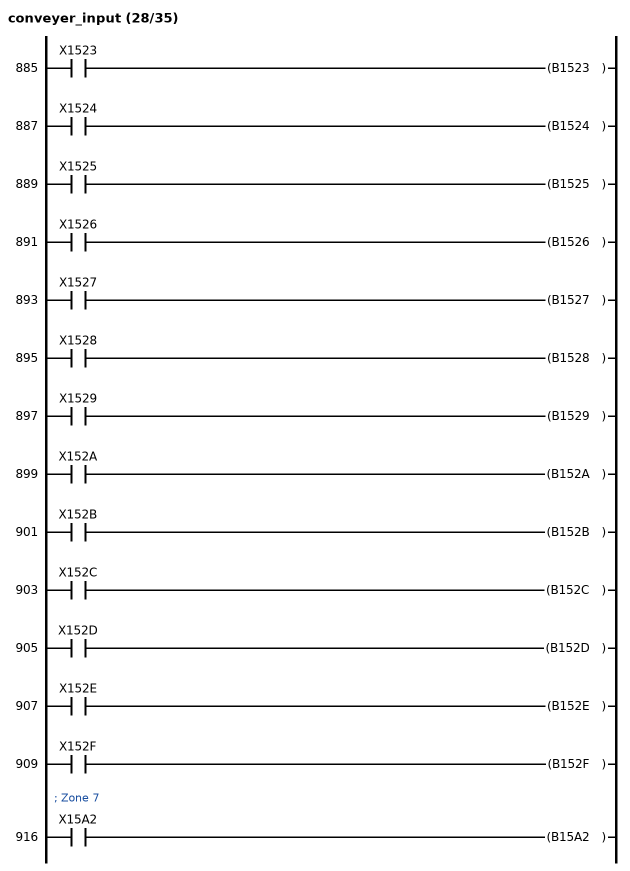
[picture p120: ladder of conveyer_input, rungs at steps 885 to 916]
885   LD      X1523
      OUT     B1523
887   LD      X1524
      OUT     B1524
889   LD      X1525
      OUT     B1525
891   LD      X1526
      OUT     B1526
893   LD      X1527
      OUT     B1527
895   LD      X1528
      OUT     B1528
897   LD      X1529
      OUT     B1529
899   LD      X152A
      OUT     B152A
901   LD      X152B
      OUT     B152B
903   LD      X152C
      OUT     B152C
905   LD      X152D
      OUT     B152D
907   LD      X152E
      OUT     B152E
909   LD      X152F
      OUT     B152F
; Zone 7
916   LD      X15A2
      OUT     B15A2
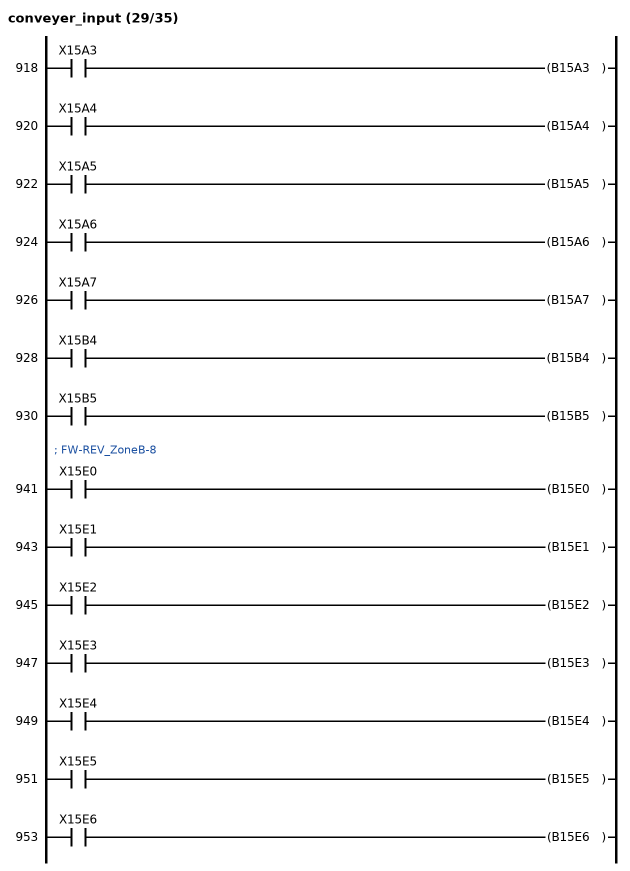
918   LD      X15A3
      OUT     B15A3
920   LD      X15A4
      OUT     B15A4
922   LD      X15A5
      OUT     B15A5
924   LD      X15A6
      OUT     B15A6
926   LD      X15A7
      OUT     B15A7
928   LD      X15B4
      OUT     B15B4
930   LD      X15B5
      OUT     B15B5
; FW-REV_ZoneB-8
941   LD      X15E0
      OUT     B15E0
943   LD      X15E1
      OUT     B15E1
945   LD      X15E2
      OUT     B15E2
947   LD      X15E3
      OUT     B15E3
949   LD      X15E4
      OUT     B15E4
951   LD      X15E5
      OUT     B15E5
953   LD      X15E6
      OUT     B15E6
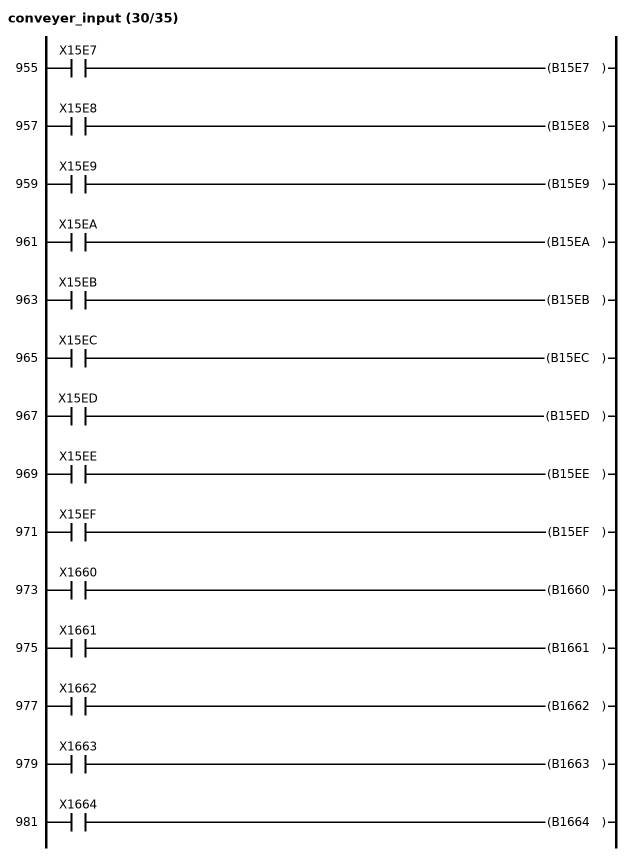
955   LD      X15E7
      OUT     B15E7
957   LD      X15E8
      OUT     B15E8
959   LD      X15E9
      OUT     B15E9
961   LD      X15EA
      OUT     B15EA
963   LD      X15EB
      OUT     B15EB
965   LD      X15EC
      OUT     B15EC
967   LD      X15ED
      OUT     B15ED
969   LD      X15EE
      OUT     B15EE
971   LD      X15EF
      OUT     B15EF
973   LD      X1660
      OUT     B1660
975   LD      X1661
      OUT     B1661
977   LD      X1662
      OUT     B1662
979   LD      X1663
      OUT     B1663
981   LD      X1664
      OUT     B1664
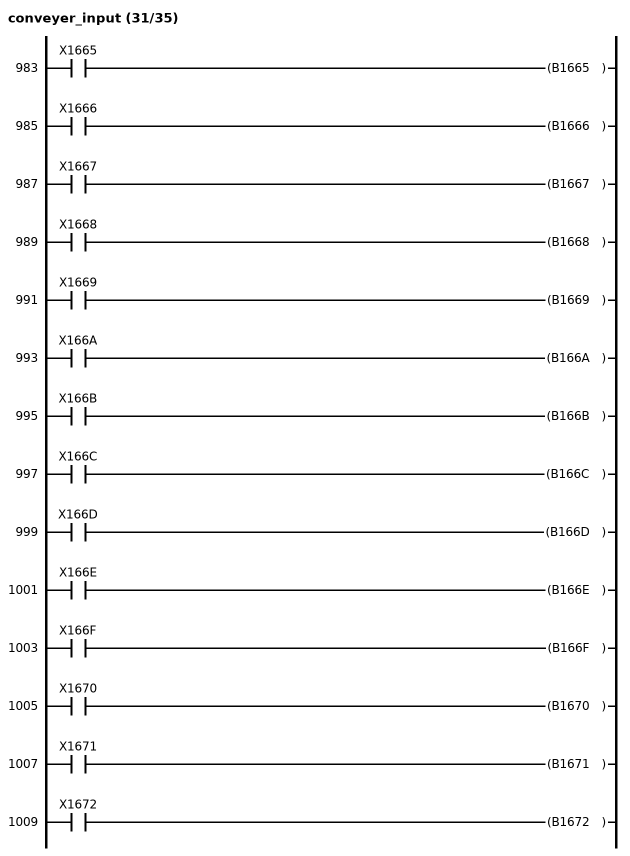
983   LD      X1665
      OUT     B1665
985   LD      X1666
      OUT     B1666
987   LD      X1667
      OUT     B1667
989   LD      X1668
      OUT     B1668
991   LD      X1669
      OUT     B1669
993   LD      X166A
      OUT     B166A
995   LD      X166B
      OUT     B166B
997   LD      X166C
      OUT     B166C
999   LD      X166D
      OUT     B166D
1001  LD      X166E
      OUT     B166E
1003  LD      X166F
      OUT     B166F
1005  LD      X1670
      OUT     B1670
1007  LD      X1671
      OUT     B1671
1009  LD      X1672
      OUT     B1672
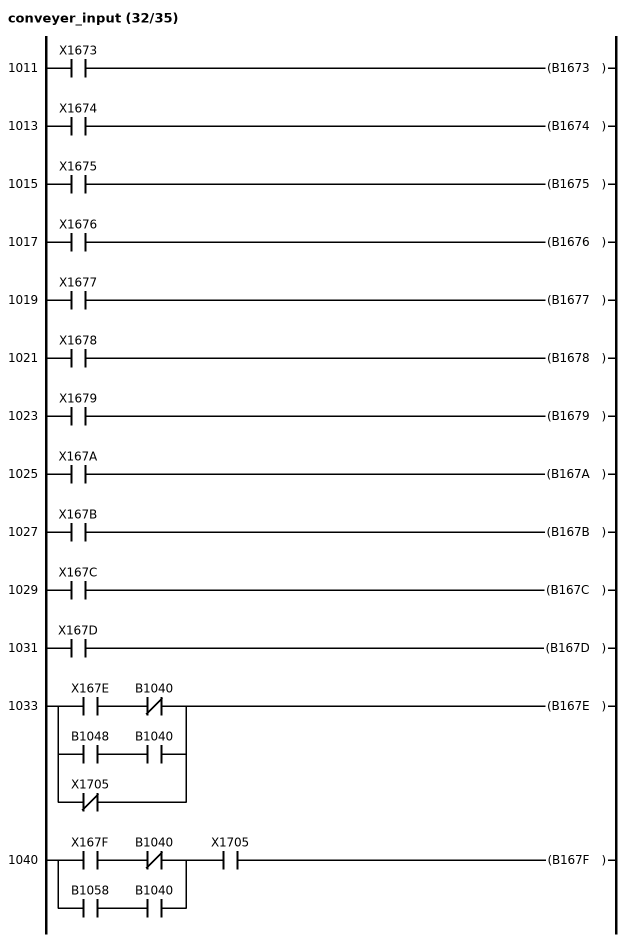
1011  LD      X1673
      OUT     B1673
1013  LD      X1674
      OUT     B1674
1015  LD      X1675
      OUT     B1675
1017  LD      X1676
      OUT     B1676
1019  LD      X1677
      OUT     B1677
1021  LD      X1678
      OUT     B1678
1023  LD      X1679
      OUT     B1679
1025  LD      X167A
      OUT     B167A
1027  LD      X167B
      OUT     B167B
1029  LD      X167C
      OUT     B167C
1031  LD      X167D
      OUT     B167D
1033  LD      X167E
      ANI     B1040
      LD      B1048
      AND     B1040
      ORB
      ORI     X1705
      OUT     B167E
1040  LD      X167F
      ANI     B1040
      LD      B1058
      AND     B1040
      ORB
      AND     X1705
      OUT     B167F
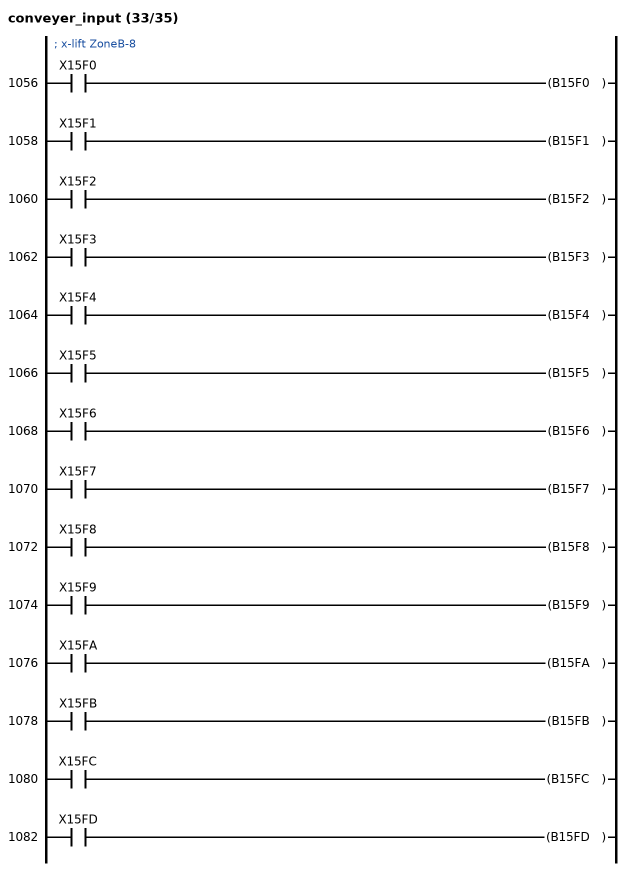
; x-lift ZoneB-8
1056  LD      X15F0
      OUT     B15F0
1058  LD      X15F1
      OUT     B15F1
1060  LD      X15F2
      OUT     B15F2
1062  LD      X15F3
      OUT     B15F3
1064  LD      X15F4
      OUT     B15F4
1066  LD      X15F5
      OUT     B15F5
1068  LD      X15F6
      OUT     B15F6
1070  LD      X15F7
      OUT     B15F7
1072  LD      X15F8
      OUT     B15F8
1074  LD      X15F9
      OUT     B15F9
1076  LD      X15FA
      OUT     B15FA
1078  LD      X15FB
      OUT     B15FB
1080  LD      X15FC
      OUT     B15FC
1082  LD      X15FD
      OUT     B15FD
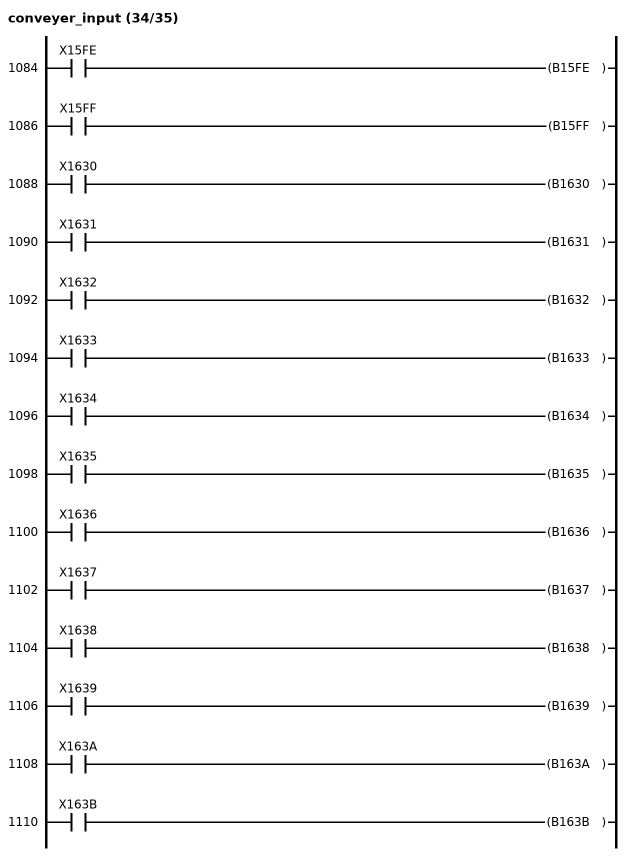
1084  LD      X15FE
      OUT     B15FE
1086  LD      X15FF
      OUT     B15FF
1088  LD      X1630
      OUT     B1630
1090  LD      X1631
      OUT     B1631
1092  LD      X1632
      OUT     B1632
1094  LD      X1633
      OUT     B1633
1096  LD      X1634
      OUT     B1634
1098  LD      X1635
      OUT     B1635
1100  LD      X1636
      OUT     B1636
1102  LD      X1637
      OUT     B1637
1104  LD      X1638
      OUT     B1638
1106  LD      X1639
      OUT     B1639
1108  LD      X163A
      OUT     B163A
1110  LD      X163B
      OUT     B163B
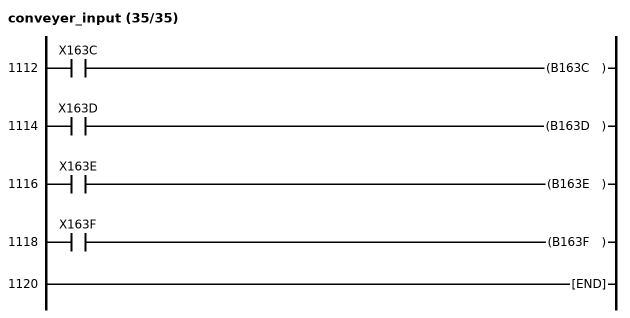
1112  LD      X163C
      OUT     B163C
1114  LD      X163D
      OUT     B163D
1116  LD      X163E
      OUT     B163E
1118  LD      X163F
      OUT     B163F
1120  END
END_PROGRAM

PROGRAM conveyor_output
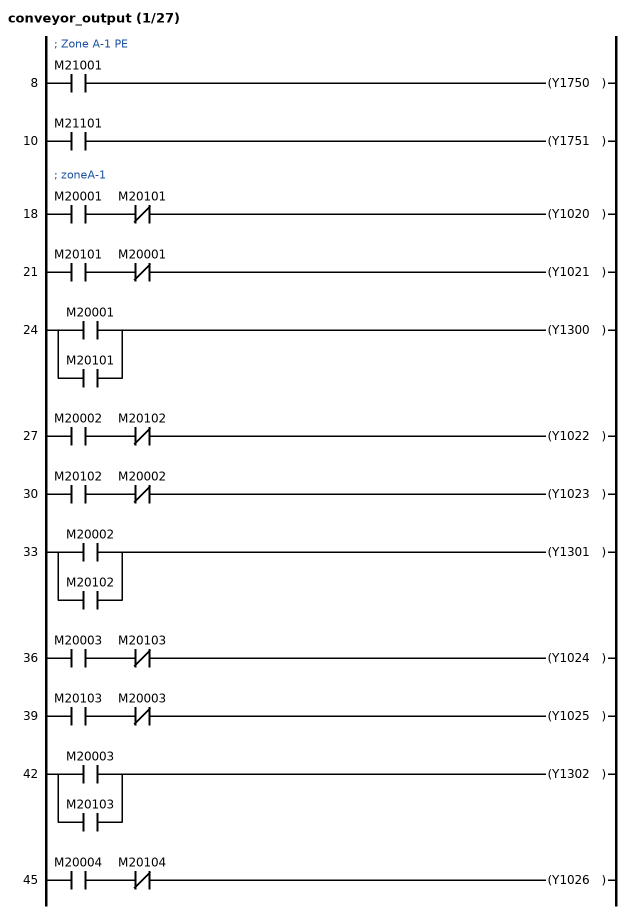
; Zone A-1 PE
8     LD      M21001
      OUT     Y1750
10    LD      M21101
      OUT     Y1751
; zoneA-1
18    LD      M20001
      ANI     M20101
      OUT     Y1020
21    LD      M20101
      ANI     M20001
      OUT     Y1021
24    LD      M20001
      OR      M20101
      OUT     Y1300
27    LD      M20002
      ANI     M20102
      OUT     Y1022
30    LD      M20102
      ANI     M20002
      OUT     Y1023
33    LD      M20002
      OR      M20102
      OUT     Y1301
36    LD      M20003
      ANI     M20103
      OUT     Y1024
39    LD      M20103
      ANI     M20003
      OUT     Y1025
42    LD      M20003
      OR      M20103
      OUT     Y1302
45    LD      M20004
      ANI     M20104
      OUT     Y1026
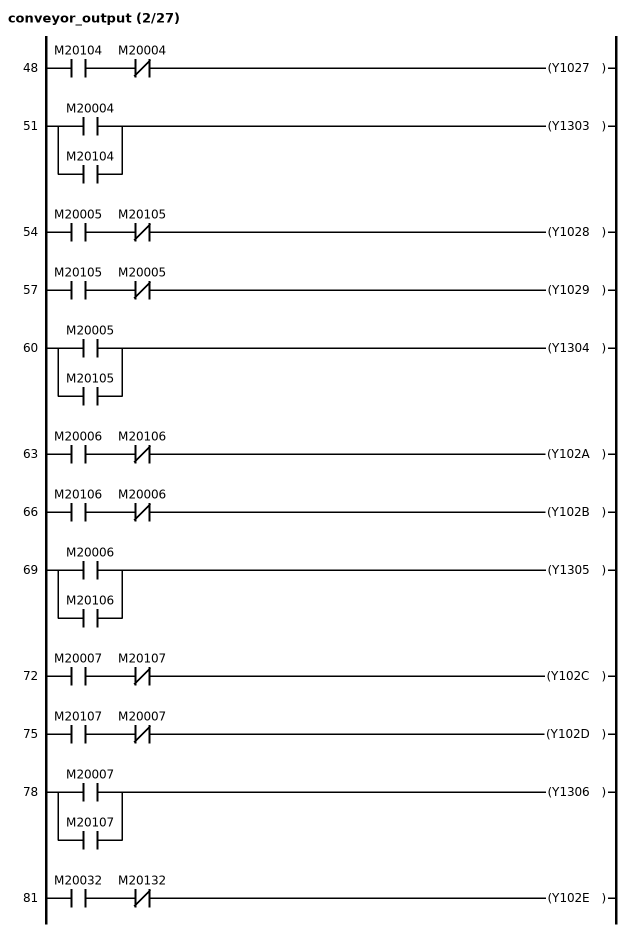
48    LD      M20104
      ANI     M20004
      OUT     Y1027
51    LD      M20004
      OR      M20104
      OUT     Y1303
54    LD      M20005
      ANI     M20105
      OUT     Y1028
57    LD      M20105
      ANI     M20005
      OUT     Y1029
60    LD      M20005
      OR      M20105
      OUT     Y1304
63    LD      M20006
      ANI     M20106
      OUT     Y102A
66    LD      M20106
      ANI     M20006
      OUT     Y102B
69    LD      M20006
      OR      M20106
      OUT     Y1305
72    LD      M20007
      ANI     M20107
      OUT     Y102C
75    LD      M20107
      ANI     M20007
      OUT     Y102D
78    LD      M20007
      OR      M20107
      OUT     Y1306
81    LD      M20032
      ANI     M20132
      OUT     Y102E
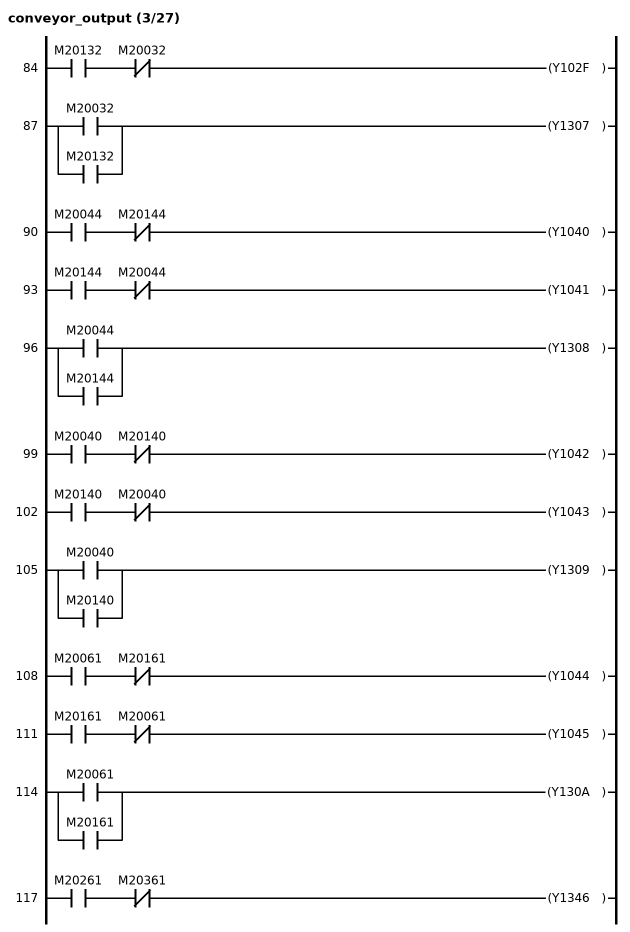
84    LD      M20132
      ANI     M20032
      OUT     Y102F
87    LD      M20032
      OR      M20132
      OUT     Y1307
90    LD      M20044
      ANI     M20144
      OUT     Y1040
93    LD      M20144
      ANI     M20044
      OUT     Y1041
96    LD      M20044
      OR      M20144
      OUT     Y1308
99    LD      M20040
      ANI     M20140
      OUT     Y1042
102   LD      M20140
      ANI     M20040
      OUT     Y1043
105   LD      M20040
      OR      M20140
      OUT     Y1309
108   LD      M20061
      ANI     M20161
      OUT     Y1044
111   LD      M20161
      ANI     M20061
      OUT     Y1045
114   LD      M20061
      OR      M20161
      OUT     Y130A
117   LD      M20261
      ANI     M20361
      OUT     Y1346
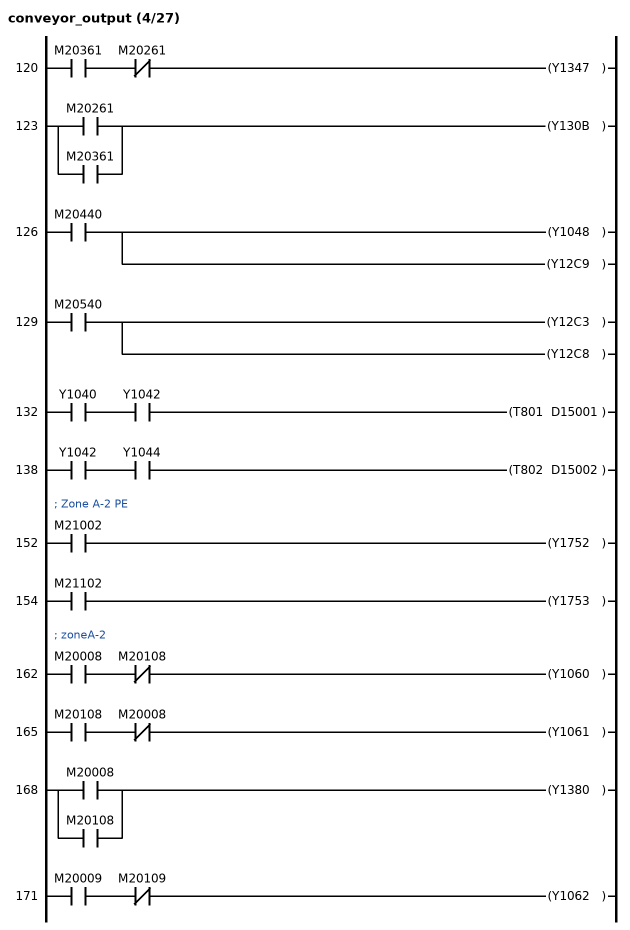
120   LD      M20361
      ANI     M20261
      OUT     Y1347
123   LD      M20261
      OR      M20361
      OUT     Y130B
126   LD      M20440
      OUT     Y1048
      OUT     Y12C9
129   LD      M20540
      OUT     Y12C3
      OUT     Y12C8
132   LD      Y1040
      AND     Y1042
      OUT     T801 D15001
138   LD      Y1042
      AND     Y1044
      OUT     T802 D15002
; Zone A-2 PE
152   LD      M21002
      OUT     Y1752
154   LD      M21102
      OUT     Y1753
; zoneA-2
162   LD      M20008
      ANI     M20108
      OUT     Y1060
165   LD      M20108
      ANI     M20008
      OUT     Y1061
168   LD      M20008
      OR      M20108
      OUT     Y1380
171   LD      M20009
      ANI     M20109
      OUT     Y1062
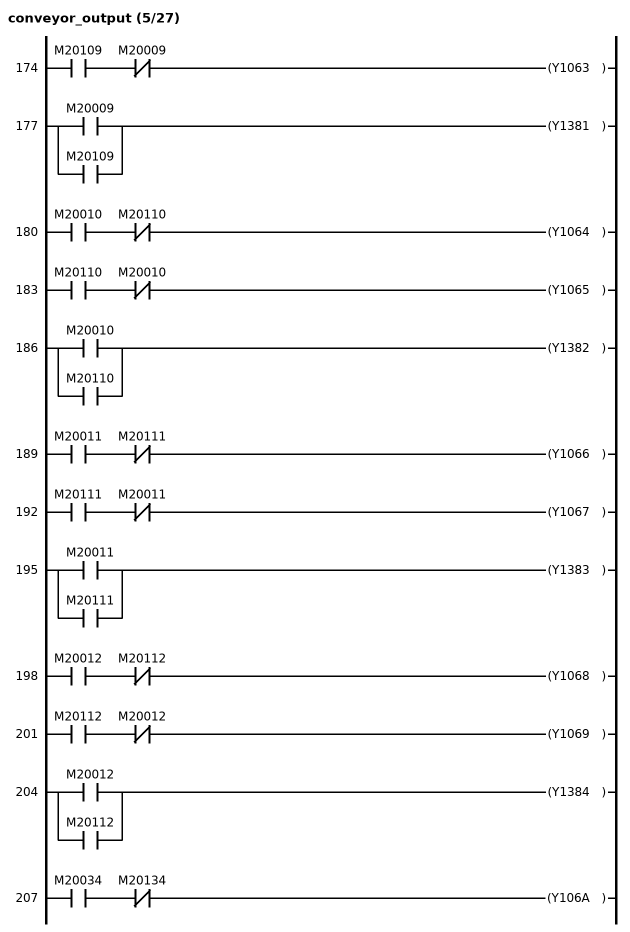
174   LD      M20109
      ANI     M20009
      OUT     Y1063
177   LD      M20009
      OR      M20109
      OUT     Y1381
180   LD      M20010
      ANI     M20110
      OUT     Y1064
183   LD      M20110
      ANI     M20010
      OUT     Y1065
186   LD      M20010
      OR      M20110
      OUT     Y1382
189   LD      M20011
      ANI     M20111
      OUT     Y1066
192   LD      M20111
      ANI     M20011
      OUT     Y1067
195   LD      M20011
      OR      M20111
      OUT     Y1383
198   LD      M20012
      ANI     M20112
      OUT     Y1068
201   LD      M20112
      ANI     M20012
      OUT     Y1069
204   LD      M20012
      OR      M20112
      OUT     Y1384
207   LD      M20034
      ANI     M20134
      OUT     Y106A
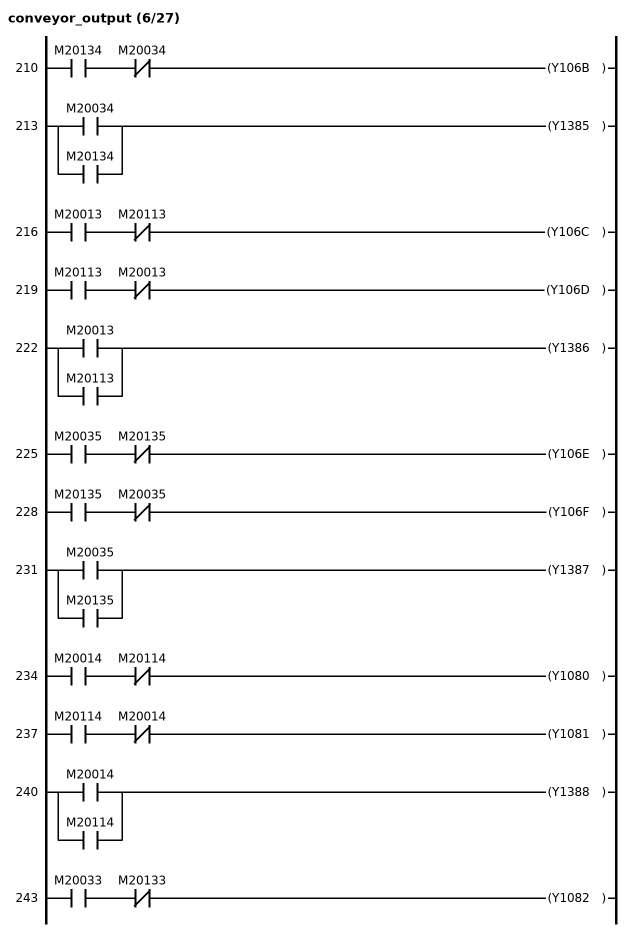
210   LD      M20134
      ANI     M20034
      OUT     Y106B
213   LD      M20034
      OR      M20134
      OUT     Y1385
216   LD      M20013
      ANI     M20113
      OUT     Y106C
219   LD      M20113
      ANI     M20013
      OUT     Y106D
222   LD      M20013
      OR      M20113
      OUT     Y1386
225   LD      M20035
      ANI     M20135
      OUT     Y106E
228   LD      M20135
      ANI     M20035
      OUT     Y106F
231   LD      M20035
      OR      M20135
      OUT     Y1387
234   LD      M20014
      ANI     M20114
      OUT     Y1080
237   LD      M20114
      ANI     M20014
      OUT     Y1081
240   LD      M20014
      OR      M20114
      OUT     Y1388
243   LD      M20033
      ANI     M20133
      OUT     Y1082
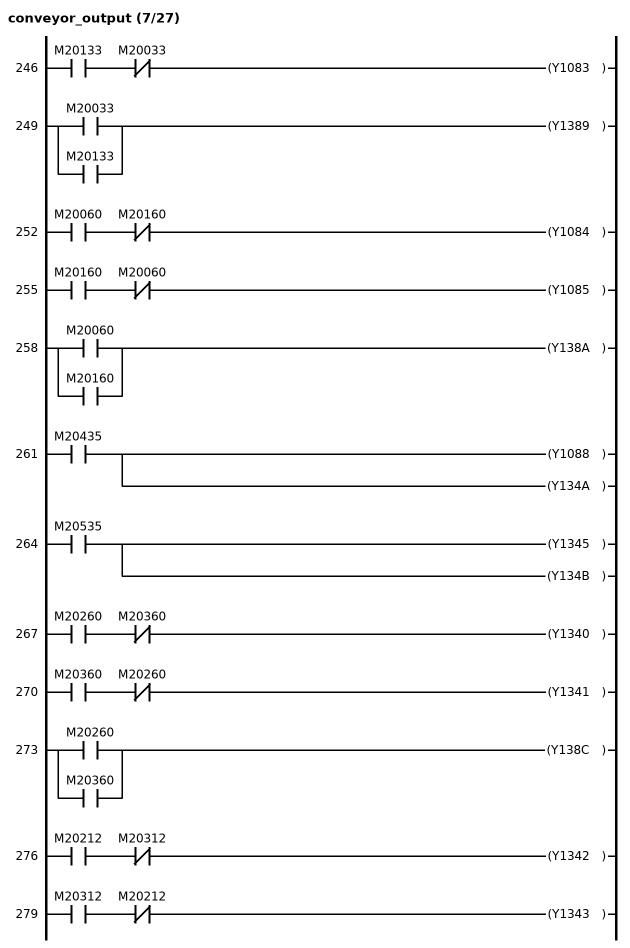
246   LD      M20133
      ANI     M20033
      OUT     Y1083
249   LD      M20033
      OR      M20133
      OUT     Y1389
252   LD      M20060
      ANI     M20160
      OUT     Y1084
255   LD      M20160
      ANI     M20060
      OUT     Y1085
258   LD      M20060
      OR      M20160
      OUT     Y138A
261   LD      M20435
      OUT     Y1088
      OUT     Y134A
264   LD      M20535
      OUT     Y1345
      OUT     Y134B
267   LD      M20260
      ANI     M20360
      OUT     Y1340
270   LD      M20360
      ANI     M20260
      OUT     Y1341
273   LD      M20260
      OR      M20360
      OUT     Y138C
276   LD      M20212
      ANI     M20312
      OUT     Y1342
279   LD      M20312
      ANI     M20212
      OUT     Y1343
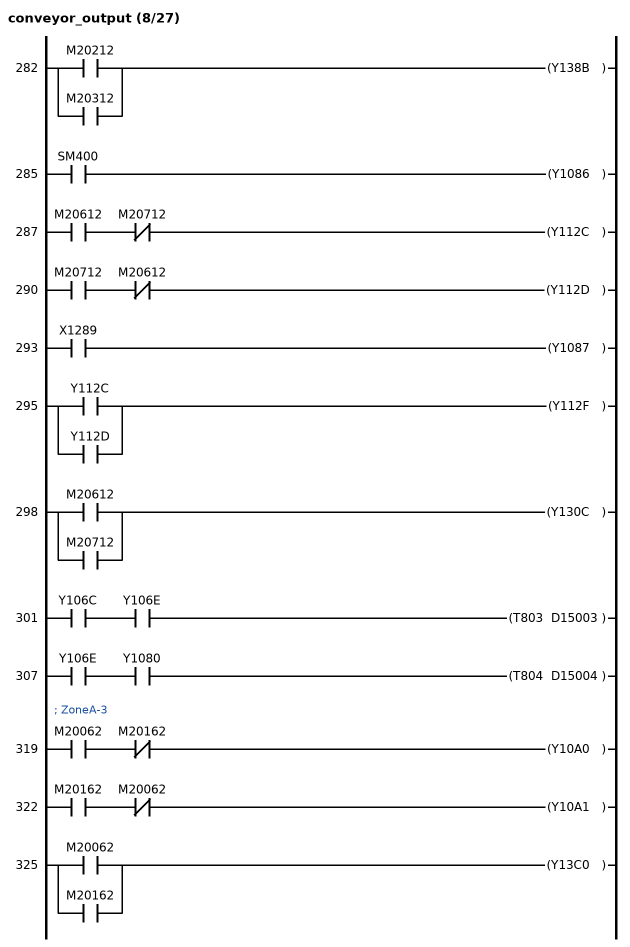
282   LD      M20212
      OR      M20312
      OUT     Y138B
285   LD      SM400
      OUT     Y1086
287   LD      M20612
      ANI     M20712
      OUT     Y112C
290   LD      M20712
      ANI     M20612
      OUT     Y112D
293   LD      X1289
      OUT     Y1087
295   LD      Y112C
      OR      Y112D
      OUT     Y112F
298   LD      M20612
      OR      M20712
      OUT     Y130C
301   LD      Y106C
      AND     Y106E
      OUT     T803 D15003
307   LD      Y106E
      AND     Y1080
      OUT     T804 D15004
; ZoneA-3
319   LD      M20062
      ANI     M20162
      OUT     Y10A0
322   LD      M20162
      ANI     M20062
      OUT     Y10A1
325   LD      M20062
      OR      M20162
      OUT     Y13C0
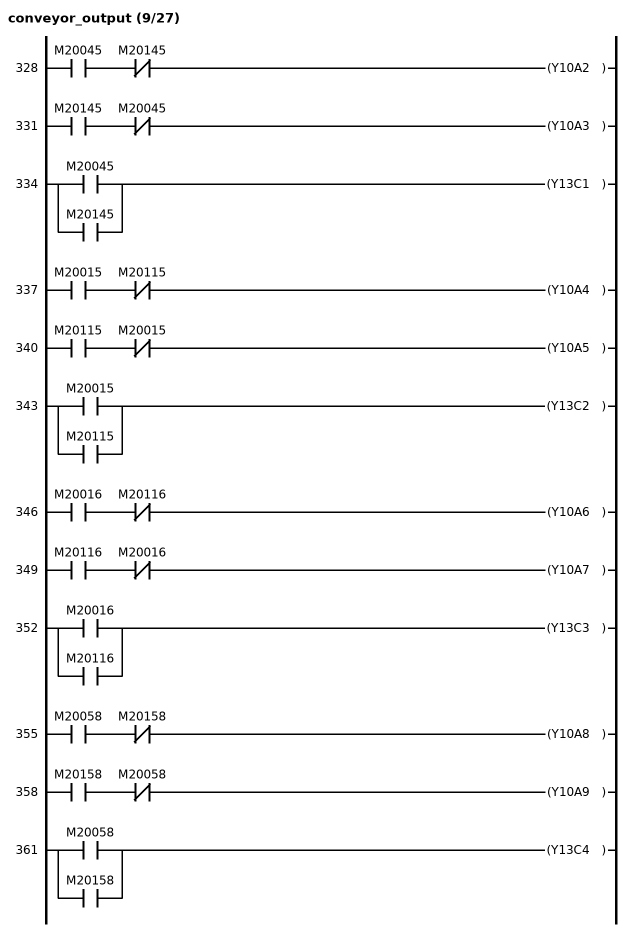
328   LD      M20045
      ANI     M20145
      OUT     Y10A2
331   LD      M20145
      ANI     M20045
      OUT     Y10A3
334   LD      M20045
      OR      M20145
      OUT     Y13C1
337   LD      M20015
      ANI     M20115
      OUT     Y10A4
340   LD      M20115
      ANI     M20015
      OUT     Y10A5
343   LD      M20015
      OR      M20115
      OUT     Y13C2
346   LD      M20016
      ANI     M20116
      OUT     Y10A6
349   LD      M20116
      ANI     M20016
      OUT     Y10A7
352   LD      M20016
      OR      M20116
      OUT     Y13C3
355   LD      M20058
      ANI     M20158
      OUT     Y10A8
358   LD      M20158
      ANI     M20058
      OUT     Y10A9
361   LD      M20058
      OR      M20158
      OUT     Y13C4
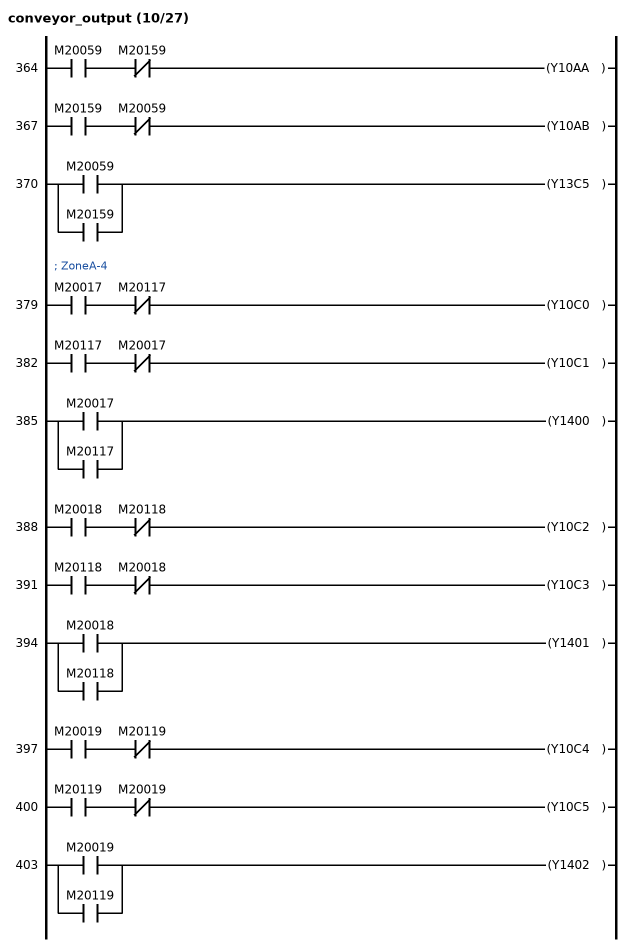
364   LD      M20059
      ANI     M20159
      OUT     Y10AA
367   LD      M20159
      ANI     M20059
      OUT     Y10AB
370   LD      M20059
      OR      M20159
      OUT     Y13C5
; ZoneA-4
379   LD      M20017
      ANI     M20117
      OUT     Y10C0
382   LD      M20117
      ANI     M20017
      OUT     Y10C1
385   LD      M20017
      OR      M20117
      OUT     Y1400
388   LD      M20018
      ANI     M20118
      OUT     Y10C2
391   LD      M20118
      ANI     M20018
      OUT     Y10C3
394   LD      M20018
      OR      M20118
      OUT     Y1401
397   LD      M20019
      ANI     M20119
      OUT     Y10C4
400   LD      M20119
      ANI     M20019
      OUT     Y10C5
403   LD      M20019
      OR      M20119
      OUT     Y1402
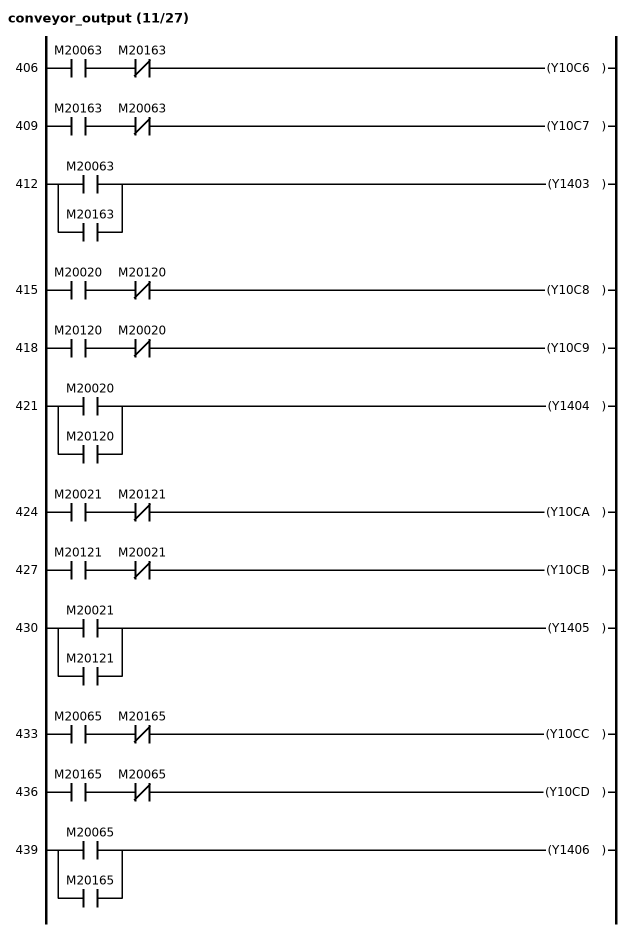
406   LD      M20063
      ANI     M20163
      OUT     Y10C6
409   LD      M20163
      ANI     M20063
      OUT     Y10C7
412   LD      M20063
      OR      M20163
      OUT     Y1403
415   LD      M20020
      ANI     M20120
      OUT     Y10C8
418   LD      M20120
      ANI     M20020
      OUT     Y10C9
421   LD      M20020
      OR      M20120
      OUT     Y1404
424   LD      M20021
      ANI     M20121
      OUT     Y10CA
427   LD      M20121
      ANI     M20021
      OUT     Y10CB
430   LD      M20021
      OR      M20121
      OUT     Y1405
433   LD      M20065
      ANI     M20165
      OUT     Y10CC
436   LD      M20165
      ANI     M20065
      OUT     Y10CD
439   LD      M20065
      OR      M20165
      OUT     Y1406
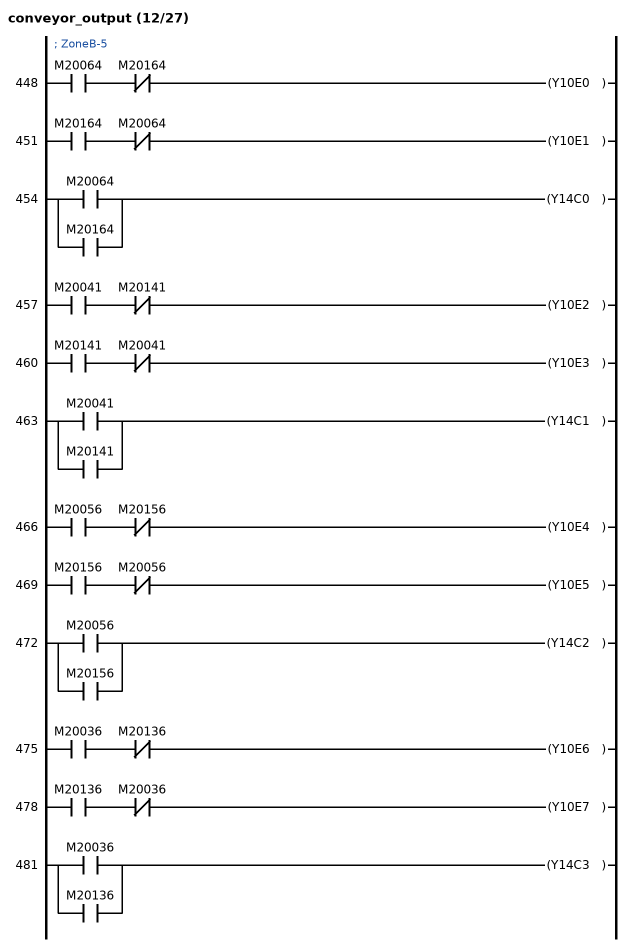
; ZoneB-5
448   LD      M20064
      ANI     M20164
      OUT     Y10E0
451   LD      M20164
      ANI     M20064
      OUT     Y10E1
454   LD      M20064
      OR      M20164
      OUT     Y14C0
457   LD      M20041
      ANI     M20141
      OUT     Y10E2
460   LD      M20141
      ANI     M20041
      OUT     Y10E3
463   LD      M20041
      OR      M20141
      OUT     Y14C1
466   LD      M20056
      ANI     M20156
      OUT     Y10E4
469   LD      M20156
      ANI     M20056
      OUT     Y10E5
472   LD      M20056
      OR      M20156
      OUT     Y14C2
475   LD      M20036
      ANI     M20136
      OUT     Y10E6
478   LD      M20136
      ANI     M20036
      OUT     Y10E7
481   LD      M20036
      OR      M20136
      OUT     Y14C3
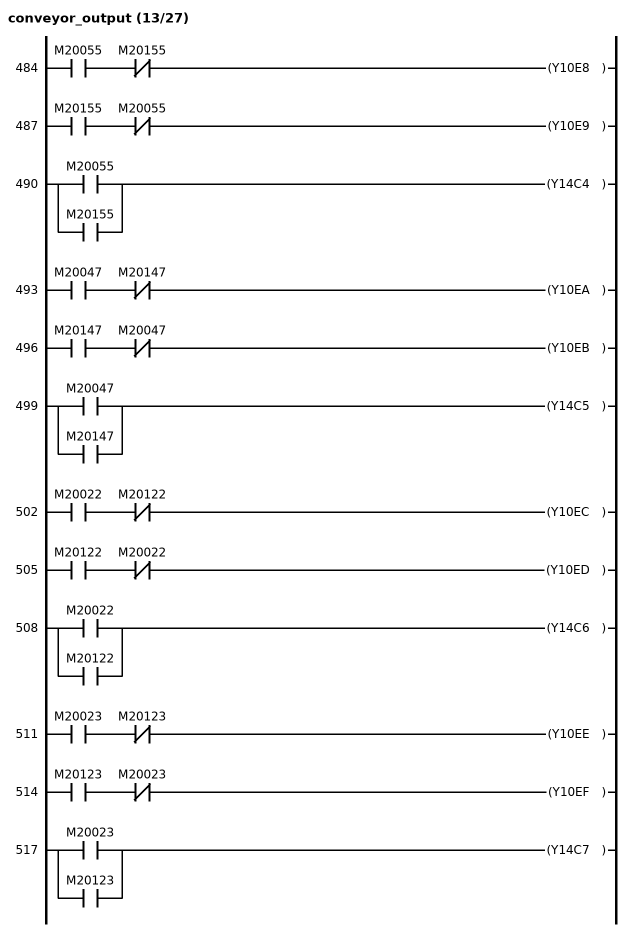
484   LD      M20055
      ANI     M20155
      OUT     Y10E8
487   LD      M20155
      ANI     M20055
      OUT     Y10E9
490   LD      M20055
      OR      M20155
      OUT     Y14C4
493   LD      M20047
      ANI     M20147
      OUT     Y10EA
496   LD      M20147
      ANI     M20047
      OUT     Y10EB
499   LD      M20047
      OR      M20147
      OUT     Y14C5
502   LD      M20022
      ANI     M20122
      OUT     Y10EC
505   LD      M20122
      ANI     M20022
      OUT     Y10ED
508   LD      M20022
      OR      M20122
      OUT     Y14C6
511   LD      M20023
      ANI     M20123
      OUT     Y10EE
514   LD      M20123
      ANI     M20023
      OUT     Y10EF
517   LD      M20023
      OR      M20123
      OUT     Y14C7
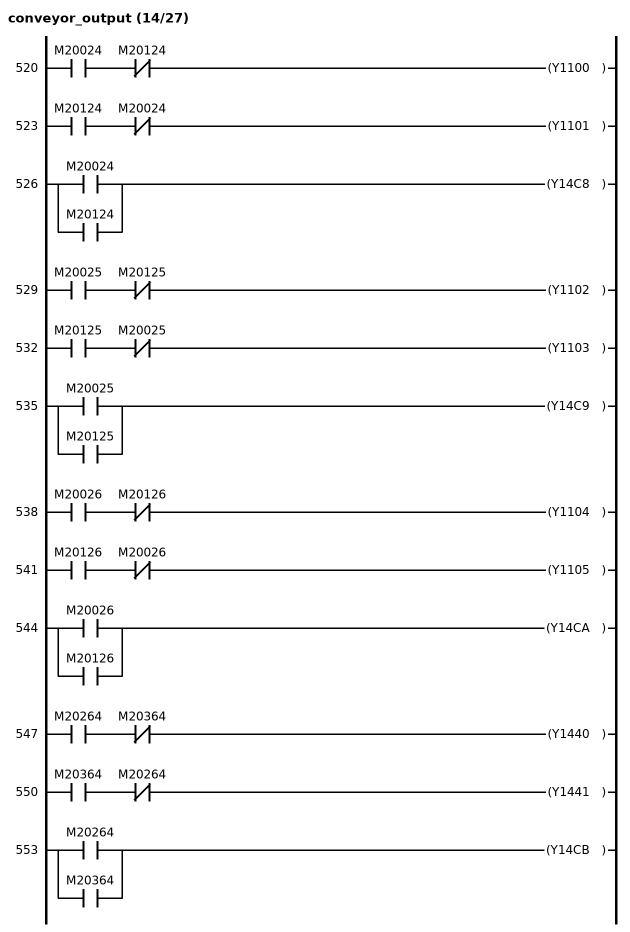
520   LD      M20024
      ANI     M20124
      OUT     Y1100
523   LD      M20124
      ANI     M20024
      OUT     Y1101
526   LD      M20024
      OR      M20124
      OUT     Y14C8
529   LD      M20025
      ANI     M20125
      OUT     Y1102
532   LD      M20125
      ANI     M20025
      OUT     Y1103
535   LD      M20025
      OR      M20125
      OUT     Y14C9
538   LD      M20026
      ANI     M20126
      OUT     Y1104
541   LD      M20126
      ANI     M20026
      OUT     Y1105
544   LD      M20026
      OR      M20126
      OUT     Y14CA
547   LD      M20264
      ANI     M20364
      OUT     Y1440
550   LD      M20364
      ANI     M20264
      OUT     Y1441
553   LD      M20264
      OR      M20364
      OUT     Y14CB
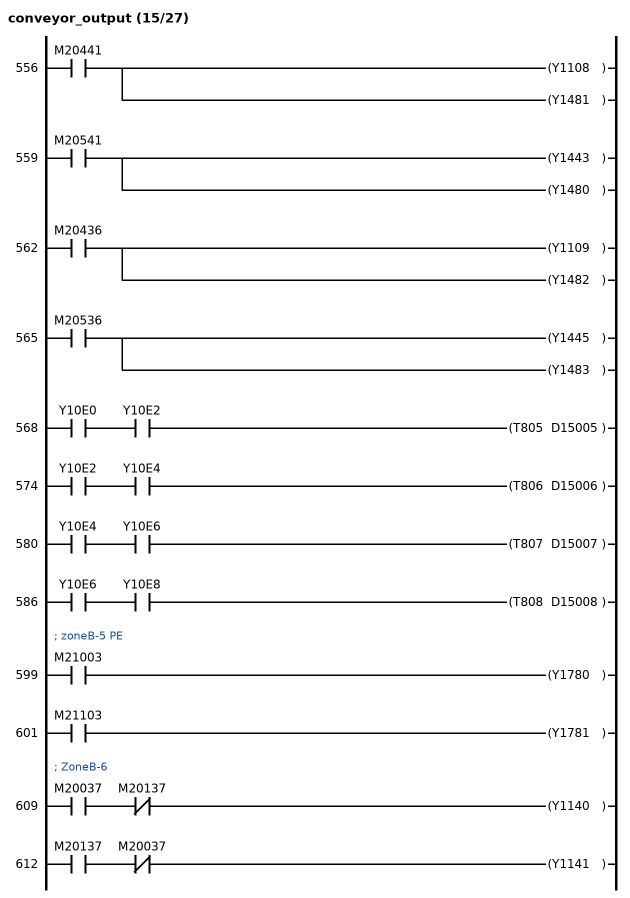
556   LD      M20441
      OUT     Y1108
      OUT     Y1481
559   LD      M20541
      OUT     Y1443
      OUT     Y1480
562   LD      M20436
      OUT     Y1109
      OUT     Y1482
565   LD      M20536
      OUT     Y1445
      OUT     Y1483
568   LD      Y10E0
      AND     Y10E2
      OUT     T805 D15005
574   LD      Y10E2
      AND     Y10E4
      OUT     T806 D15006
580   LD      Y10E4
      AND     Y10E6
      OUT     T807 D15007
586   LD      Y10E6
      AND     Y10E8
      OUT     T808 D15008
; zoneB-5 PE
599   LD      M21003
      OUT     Y1780
601   LD      M21103
      OUT     Y1781
; ZoneB-6
609   LD      M20037
      ANI     M20137
      OUT     Y1140
612   LD      M20137
      ANI     M20037
      OUT     Y1141
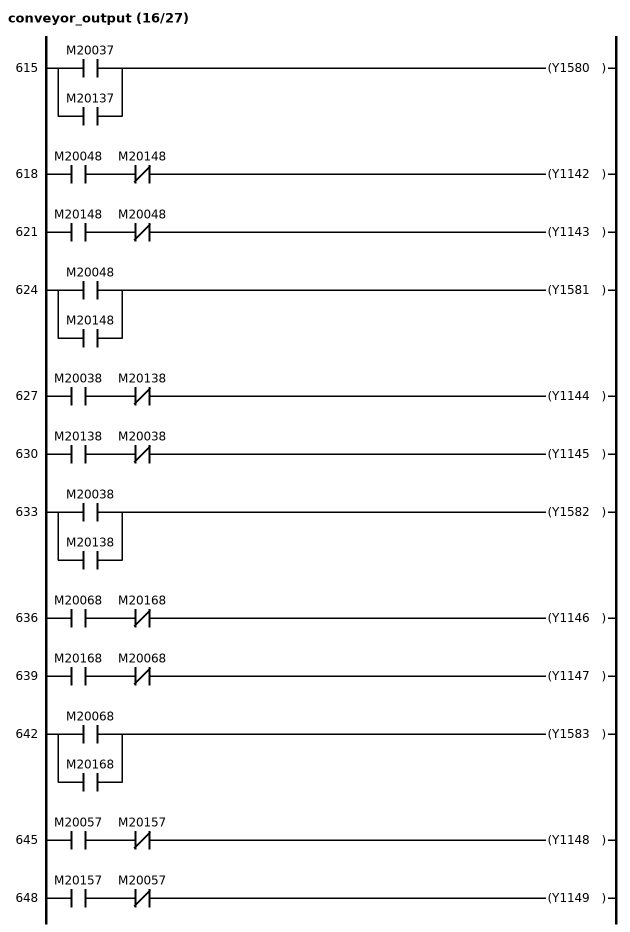
615   LD      M20037
      OR      M20137
      OUT     Y1580
618   LD      M20048
      ANI     M20148
      OUT     Y1142
621   LD      M20148
      ANI     M20048
      OUT     Y1143
624   LD      M20048
      OR      M20148
      OUT     Y1581
627   LD      M20038
      ANI     M20138
      OUT     Y1144
630   LD      M20138
      ANI     M20038
      OUT     Y1145
633   LD      M20038
      OR      M20138
      OUT     Y1582
636   LD      M20068
      ANI     M20168
      OUT     Y1146
639   LD      M20168
      ANI     M20068
      OUT     Y1147
642   LD      M20068
      OR      M20168
      OUT     Y1583
645   LD      M20057
      ANI     M20157
      OUT     Y1148
648   LD      M20157
      ANI     M20057
      OUT     Y1149
